{attribute 'qualified_only'}
VAR_GLOBAL
	active		: BOOL;
	generate	: BOOL;
	shift		: BOOL;
	delete		: BOOL;
	safetyNOK	: BOOL;
	fault		: BOOL;
END_VAR

(* stored: Version 1.1.0.1
   GVL SIM: Id {51c77c69-2f5c-4ecd-a822-0cf4fc2a5f43} *)
